(* CFC diagram, written out as Structured Text *)
(* KNX Sending interval *)
(* KNX Master *)
Interval(IN := Interval.Q);
_ADD9_OUT := BOOL_TO_INT(Interval.Q) + i;
i := _ADD9_OUT;
_GT15_OUT := i > 83;
_MOVE19_OUT := MOVE(EN := _GT15_OUT, IN := 0, ENO => _MOVE19_ENO);
IF _MOVE19_ENO THEN i := _MOVE19_OUT; END_IF;
KNX_master_1(I_Port := IoConfig_Globals.KNX_EIB_TP1_Interface, bPortKNX := 1);
STLV59_563.STLV59_A_563_KNX_Card_1_Status := KNX_master_1.sStatus = 'OK';
(* Rom 001 *)
(* RB601_V *)
(* RB601_HVAC *)
M1_001_001_RB601_V(bPortKNX := 1, dwIndex_DPT := 1, typDPT := typDPT);
_MOVE46_OUT := MOVE(EN := M1_001_001_RB601_V.xUpdate_PLC, IN := M1_001_001_RB601_V.xSwitch_OUT, ENO => _MOVE46_ENO);
IF _MOVE46_ENO THEN STLV59_563.STLV59_A_563_001.RB601_V := _MOVE46_OUT; END_IF;
M1_002_001_RB601_HVAC(bPortKNX := 1, dwIndex_DPT := 2, typDPT := typDPT);
_MOVE59_OUT := MOVE(EN := M1_002_001_RB601_HVAC.xUpdate_PLC, IN := M1_002_001_RB601_HVAC.xSwitch_OUT, ENO => _MOVE59_ENO);
IF _MOVE59_ENO THEN STLV59_563.STLV59_A_563_001.RB601_HVAC := _MOVE59_OUT; END_IF;
(* RT601_CT *)
(* RY601_CV *)
M1_003_001_RT601_CT(bPortKNX := 1, dwIndex_DPT := 3, typDPT := typDPT);
_MOVE72_OUT := MOVE(EN := M1_003_001_RT601_CT.xUpdate_PLC, IN := M1_003_001_RT601_CT.rValue_OUT, ENO => _MOVE72_ENO);
IF _MOVE72_ENO THEN STLV59_563.STLV59_A_563_001.RT601_CT := _MOVE72_OUT; END_IF;
M1_004_001_RY601_CV(bPortKNX := 1, dwIndex_DPT := 4, typDPT := typDPT);
_MOVE85_OUT := MOVE(EN := M1_004_001_RY601_CV.xUpdate_PLC, IN := M1_004_001_RY601_CV.rValue_OUT, ENO => _MOVE85_ENO);
IF _MOVE85_ENO THEN STLV59_563.STLV59_A_563_001.RY601_CV := _MOVE85_OUT; END_IF;
(* LH601_OP *)
(* LH601_CMD *)
M1_005_001_LH601_OP(bPortKNX := 1, dwIndex_DPT := 5, rValue_IN := STLV59_563.STLV59_A_563_001.LH601_OP, xUpdate_KNX := i = 0, typDPT := typDPT);
M1_006_001_LH601_CMD(bPortKNX := 1, dwIndex_DPT := 6, xSwitch_IN := STLV59_563.STLV59_A_563_001.LH601_CMD, xUpdate_KNX := i = 1, typDPT := typDPT);
(* LC601_OP *)
(* LC601_CMD *)
M1_007_001_LC601_OP(bPortKNX := 1, dwIndex_DPT := 7, rValue_IN := STLV59_563.STLV59_A_563_001.LC601_OP, xUpdate_KNX := i = 2, typDPT := typDPT);
M1_008_001_LC601_CMD(bPortKNX := 1, dwIndex_DPT := 8, xSwitch_IN := STLV59_563.STLV59_A_563_001.LC601_CMD, xUpdate_KNX := i = 3, typDPT := typDPT);
(* Rom 002 *)
(* RB601_V *)
(* RB602_V *)
M1_009_002_RB601_V(bPortKNX := 1, dwIndex_DPT := 9, typDPT := typDPT);
_MOVE163_OUT := MOVE(EN := M1_009_002_RB601_V.xUpdate_PLC, IN := M1_009_002_RB601_V.xSwitch_OUT, ENO => _MOVE163_ENO);
IF _MOVE163_ENO THEN STLV59_563.STLV59_A_563_002.RB601_V := _MOVE163_OUT; END_IF;
M1_0010_002_RB602_V(bPortKNX := 1, dwIndex_DPT := 10, typDPT := typDPT);
_MOVE176_OUT := MOVE(EN := M1_0010_002_RB602_V.xUpdate_PLC, IN := M1_0010_002_RB602_V.xSwitch_OUT, ENO => _MOVE176_ENO);
IF _MOVE176_ENO THEN STLV59_563.STLV59_A_563_002.RB602_V := _MOVE176_OUT; END_IF;
(* RB601_HVAC *)
(* RB602_HVAC *)
M1_011_002_RB601_HVAC(bPortKNX := 1, dwIndex_DPT := 11, typDPT := typDPT);
_MOVE189_OUT := MOVE(EN := M1_011_002_RB601_HVAC.xUpdate_PLC, IN := M1_011_002_RB601_HVAC.xSwitch_OUT, ENO => _MOVE189_ENO);
IF _MOVE189_ENO THEN STLV59_563.STLV59_A_563_002.RB601_HVAC := _MOVE189_OUT; END_IF;
M1_012_002_RB602_HVAC(bPortKNX := 1, dwIndex_DPT := 12, typDPT := typDPT);
_MOVE202_OUT := MOVE(EN := M1_012_002_RB602_HVAC.xUpdate_PLC, IN := M1_012_002_RB602_HVAC.xSwitch_OUT, ENO => _MOVE202_ENO);
IF _MOVE202_ENO THEN STLV59_563.STLV59_A_563_002.RB602_HVAC := _MOVE202_OUT; END_IF;
(* RT601_CT *)
(* RY601_CV *)
M1_013_002_RT601_CT(bPortKNX := 1, dwIndex_DPT := 13, typDPT := typDPT);
_MOVE215_OUT := MOVE(EN := M1_013_002_RT601_CT.xUpdate_PLC, IN := M1_013_002_RT601_CT.rValue_OUT, ENO => _MOVE215_ENO);
IF _MOVE215_ENO THEN STLV59_563.STLV59_A_563_002.RT601_CT := _MOVE215_OUT; END_IF;
M1_014_002_RY601_CV(bPortKNX := 1, dwIndex_DPT := 14, typDPT := typDPT);
_MOVE228_OUT := MOVE(EN := M1_014_002_RY601_CV.xUpdate_PLC, IN := M1_014_002_RY601_CV.rValue_OUT, ENO => _MOVE228_ENO);
IF _MOVE228_ENO THEN STLV59_563.STLV59_A_563_002.RY601_CV := _MOVE228_OUT; END_IF;
(* LH601_OP *)
(* LH601_CMD *)
M1_015_002_LH601_OP(bPortKNX := 1, dwIndex_DPT := 15, rValue_IN := STLV59_563.STLV59_A_563_002.LH601_OP, xUpdate_KNX := i = 4, typDPT := typDPT);
M1_016_002_LH601_CMD(bPortKNX := 1, dwIndex_DPT := 16, xSwitch_IN := STLV59_563.STLV59_A_563_002.LH601_CMD, xUpdate_KNX := i = 5, typDPT := typDPT);
(* LC601_OP *)
(* LC601_CMD *)
M1_017_002_LC601_OP(bPortKNX := 1, dwIndex_DPT := 17, rValue_IN := STLV59_563.STLV59_A_563_002.LC601_OP, xUpdate_KNX := i = 6, typDPT := typDPT);
M1_018_002_LC601_CMD(bPortKNX := 1, dwIndex_DPT := 18, xSwitch_IN := STLV59_563.STLV59_A_563_002.LC601_CMD, xUpdate_KNX := i = 7, typDPT := typDPT);
(* Rom 003 *)
(* RB601_V *)
(* RB601_HVAC *)
M1_019_003_RB601_V(bPortKNX := 1, dwIndex_DPT := 19, typDPT := typDPT);
_MOVE306_OUT := MOVE(EN := M1_019_003_RB601_V.xUpdate_PLC, IN := M1_019_003_RB601_V.xSwitch_OUT, ENO => _MOVE306_ENO);
IF _MOVE306_ENO THEN STLV59_563.STLV59_A_563_003.RB601_V := _MOVE306_OUT; END_IF;
M1_020_003_RB601_HVAC(bPortKNX := 1, dwIndex_DPT := 20, typDPT := typDPT);
_MOVE319_OUT := MOVE(EN := M1_020_003_RB601_HVAC.xUpdate_PLC, IN := M1_020_003_RB601_HVAC.xSwitch_OUT, ENO => _MOVE319_ENO);
IF _MOVE319_ENO THEN STLV59_563.STLV59_A_563_003.RB601_HVAC := _MOVE319_OUT; END_IF;
(* RT601_CT *)
(* RT602_CT *)
M1_021_003_RT601_CT(bPortKNX := 1, dwIndex_DPT := 21, typDPT := typDPT);
_MOVE332_OUT := MOVE(EN := M1_021_003_RT601_CT.xUpdate_PLC, IN := M1_021_003_RT601_CT.rValue_OUT, ENO => _MOVE332_ENO);
IF _MOVE332_ENO THEN STLV59_563.STLV59_A_563_003.RT601_CT := _MOVE332_OUT; END_IF;
M1_022_003_RT602_CT(bPortKNX := 1, dwIndex_DPT := 22, typDPT := typDPT);
_MOVE345_OUT := MOVE(EN := M1_022_003_RT602_CT.xUpdate_PLC, IN := M1_022_003_RT602_CT.rValue_OUT, ENO => _MOVE345_ENO);
IF _MOVE345_ENO THEN STLV59_563.STLV59_A_563_003.RT602_CT := _MOVE345_OUT; END_IF;
(* RY601_CV *)
(* LH601_OP *)
M1_023_003_RY601_CV(bPortKNX := 1, dwIndex_DPT := 23, typDPT := typDPT);
_MOVE358_OUT := MOVE(EN := M1_023_003_RY601_CV.xUpdate_PLC, IN := M1_023_003_RY601_CV.rValue_OUT, ENO => _MOVE358_ENO);
IF _MOVE358_ENO THEN STLV59_563.STLV59_A_563_003.RY601_CV := _MOVE358_OUT; END_IF;
M1_024_003_LH601_OP(bPortKNX := 1, dwIndex_DPT := 24, rValue_IN := STLV59_563.STLV59_A_563_003.LH601_OP, xUpdate_KNX := i = 8, typDPT := typDPT);
(* LH601_CMD *)
(* LC601_OP *)
M1_025_003_LH601_CMD(bPortKNX := 1, dwIndex_DPT := 25, xSwitch_IN := STLV59_563.STLV59_A_563_003.LH601_CMD, xUpdate_KNX := i = 9, typDPT := typDPT);
M1_026_003_LC601_OP(bPortKNX := 1, dwIndex_DPT := 26, rValue_IN := STLV59_563.STLV59_A_563_003.LC601_OP, xUpdate_KNX := i = 10, typDPT := typDPT);
(* LC601_CMD *)
M1_027_003_LC601_CMD(bPortKNX := 1, dwIndex_DPT := 27, xSwitch_IN := STLV59_563.STLV59_A_563_003.LC601_CMD, xUpdate_KNX := i = 11, typDPT := typDPT);
(* Rom 004 *)
(* RB601_V *)
(* RB601_HVAC *)
M1_028_004_RB601_V(bPortKNX := 1, dwIndex_DPT := 28, typDPT := typDPT);
_MOVE436_OUT := MOVE(EN := M1_028_004_RB601_V.xUpdate_PLC, IN := M1_028_004_RB601_V.xSwitch_OUT, ENO => _MOVE436_ENO);
IF _MOVE436_ENO THEN STLV59_563.STLV59_A_563_004.RB601_V := _MOVE436_OUT; END_IF;
M1_029_004_RB601_HVAC(bPortKNX := 1, dwIndex_DPT := 29, typDPT := typDPT);
_MOVE449_OUT := MOVE(EN := M1_029_004_RB601_HVAC.xUpdate_PLC, IN := M1_029_004_RB601_HVAC.xSwitch_OUT, ENO => _MOVE449_ENO);
IF _MOVE449_ENO THEN STLV59_563.STLV59_A_563_004.RB601_HVAC := _MOVE449_OUT; END_IF;
(* RT601_CT *)
(* RY601_CV *)
M1_030_004_RT601_CT(bPortKNX := 1, dwIndex_DPT := 30, typDPT := typDPT);
_MOVE462_OUT := MOVE(EN := M1_030_004_RT601_CT.xUpdate_PLC, IN := M1_030_004_RT601_CT.rValue_OUT, ENO => _MOVE462_ENO);
IF _MOVE462_ENO THEN STLV59_563.STLV59_A_563_004.RT601_CT := _MOVE462_OUT; END_IF;
M1_031_004_RY601_CV(bPortKNX := 1, dwIndex_DPT := 31, typDPT := typDPT);
_MOVE475_OUT := MOVE(EN := M1_031_004_RY601_CV.xUpdate_PLC, IN := M1_031_004_RY601_CV.rValue_OUT, ENO => _MOVE475_ENO);
IF _MOVE475_ENO THEN STLV59_563.STLV59_A_563_004.RY601_CV := _MOVE475_OUT; END_IF;
(* RY602_CV *)
(* LH601_OP *)
M1_032_004_RY602_CV(bPortKNX := 1, dwIndex_DPT := 32, typDPT := typDPT);
_MOVE488_OUT := MOVE(EN := M1_032_004_RY602_CV.xUpdate_PLC, IN := M1_032_004_RY602_CV.rValue_OUT, ENO => _MOVE488_ENO);
IF _MOVE488_ENO THEN STLV59_563.STLV59_A_563_004.RY602_CV := _MOVE488_OUT; END_IF;
M1_033_004_LH601_OP(bPortKNX := 1, dwIndex_DPT := 33, rValue_IN := STLV59_563.STLV59_A_563_004.LH601_OP, xUpdate_KNX := i = 12, typDPT := typDPT);
(* LH601_CMD *)
(* LC601_OP *)
M1_034_004_LH601_CMD(bPortKNX := 1, dwIndex_DPT := 34, xSwitch_IN := STLV59_563.STLV59_A_563_004.LH601_CMD, xUpdate_KNX := i = 13, typDPT := typDPT);
M1_035_004_LC601_OP(bPortKNX := 1, dwIndex_DPT := 35, rValue_IN := STLV59_563.STLV59_A_563_004.LC601_OP, xUpdate_KNX := i = 14, typDPT := typDPT);
(* LC601_CMD *)
M1_036_004_LC601_CMD(bPortKNX := 1, dwIndex_DPT := 36, xSwitch_IN := STLV59_563.STLV59_A_563_004.LC601_CMD, xUpdate_KNX := i = 15, typDPT := typDPT);
(* Rom 005 *)
(* RB601_V *)
(* RB601_HVAC *)
M1_037_005_RB601_V(bPortKNX := 1, dwIndex_DPT := 37, typDPT := typDPT);
_MOVE566_OUT := MOVE(EN := M1_037_005_RB601_V.xUpdate_PLC, IN := M1_037_005_RB601_V.xSwitch_OUT, ENO => _MOVE566_ENO);
IF _MOVE566_ENO THEN STLV59_563.STLV59_A_563_005.RB601_V := _MOVE566_OUT; END_IF;
M1_038_005_RB601_HVAC(bPortKNX := 1, dwIndex_DPT := 38, typDPT := typDPT);
_MOVE579_OUT := MOVE(EN := M1_038_005_RB601_HVAC.xUpdate_PLC, IN := M1_038_005_RB601_HVAC.xSwitch_OUT, ENO => _MOVE579_ENO);
IF _MOVE579_ENO THEN STLV59_563.STLV59_A_563_005.RB601_HVAC := _MOVE579_OUT; END_IF;
(* RT601_CT *)
(* RY601_CV *)
M1_039_005_RT601_CT(bPortKNX := 1, dwIndex_DPT := 39, typDPT := typDPT);
_MOVE592_OUT := MOVE(EN := M1_039_005_RT601_CT.xUpdate_PLC, IN := M1_039_005_RT601_CT.rValue_OUT, ENO => _MOVE592_ENO);
IF _MOVE592_ENO THEN STLV59_563.STLV59_A_563_005.RT601_CT := _MOVE592_OUT; END_IF;
M1_040_005_RY601_CV(bPortKNX := 1, dwIndex_DPT := 40, typDPT := typDPT);
_MOVE605_OUT := MOVE(EN := M1_040_005_RY601_CV.xUpdate_PLC, IN := M1_040_005_RY601_CV.rValue_OUT, ENO => _MOVE605_ENO);
IF _MOVE605_ENO THEN STLV59_563.STLV59_A_563_005.RY601_CV := _MOVE605_OUT; END_IF;
(* LH601_OP *)
(* LH602_OP *)
M1_041_005_LH601_OP(bPortKNX := 1, dwIndex_DPT := 41, rValue_IN := STLV59_563.STLV59_A_563_005.LH601_OP, xUpdate_KNX := i = 16, typDPT := typDPT);
M1_042_005_LH602_OP(bPortKNX := 1, dwIndex_DPT := 42, rValue_IN := STLV59_563.STLV59_A_563_005.LH602_OP, xUpdate_KNX := i = 17, typDPT := typDPT);
(* LH601_CMD *)
(* LC601_OP *)
M1_043_005_LH601_CMD(bPortKNX := 1, dwIndex_DPT := 43, xSwitch_IN := STLV59_563.STLV59_A_563_005.LH601_CMD, xUpdate_KNX := i = 18, typDPT := typDPT);
M1_044_005_LC601_OP(bPortKNX := 1, dwIndex_DPT := 44, rValue_IN := STLV59_563.STLV59_A_563_005.LC601_OP, xUpdate_KNX := i = 19, typDPT := typDPT);
(* LC601_CMD *)
M1_045_005_LC601_CMD(bPortKNX := 1, dwIndex_DPT := 45, xSwitch_IN := STLV59_563.STLV59_A_563_005.LC601_CMD, xUpdate_KNX := i = 20, typDPT := typDPT);
(* Rom 006 *)
(* RB601_V *)
(* RB601_HVAC *)
M1_046_006_RB601_V(bPortKNX := 1, dwIndex_DPT := 46, typDPT := typDPT);
_MOVE699_OUT := MOVE(EN := M1_046_006_RB601_V.xUpdate_PLC, IN := M1_046_006_RB601_V.xSwitch_OUT, ENO => _MOVE699_ENO);
IF _MOVE699_ENO THEN STLV59_563.STLV59_A_563_006.RB601_V := _MOVE699_OUT; END_IF;
M1_047_006_RB601_HVAC(bPortKNX := 1, dwIndex_DPT := 47, typDPT := typDPT);
_MOVE712_OUT := MOVE(EN := M1_047_006_RB601_HVAC.xUpdate_PLC, IN := M1_047_006_RB601_HVAC.xSwitch_OUT, ENO => _MOVE712_ENO);
IF _MOVE712_ENO THEN STLV59_563.STLV59_A_563_006.RB601_HVAC := _MOVE712_OUT; END_IF;
(* RT601_CT *)
(* RY601_CV *)
M1_048_006_RT601_CT(bPortKNX := 1, dwIndex_DPT := 48, typDPT := typDPT);
_MOVE725_OUT := MOVE(EN := M1_048_006_RT601_CT.xUpdate_PLC, IN := M1_048_006_RT601_CT.rValue_OUT, ENO => _MOVE725_ENO);
IF _MOVE725_ENO THEN STLV59_563.STLV59_A_563_006.RT601_CT := _MOVE725_OUT; END_IF;
M1_049_006_RY601_CV(bPortKNX := 1, dwIndex_DPT := 49, typDPT := typDPT);
_MOVE738_OUT := MOVE(EN := M1_049_006_RY601_CV.xUpdate_PLC, IN := M1_049_006_RY601_CV.rValue_OUT, ENO => _MOVE738_ENO);
IF _MOVE738_ENO THEN STLV59_563.STLV59_A_563_006.RY601_CV := _MOVE738_OUT; END_IF;
(* LH601_OP *)
(* LH601_CMD *)
M1_050_006_LH601_OP(bPortKNX := 1, dwIndex_DPT := 50, rValue_IN := STLV59_563.STLV59_A_563_006.LH601_OP, xUpdate_KNX := i = 21, typDPT := typDPT);
M1_051_006_LH601_CMD(bPortKNX := 1, dwIndex_DPT := 51, xSwitch_IN := STLV59_563.STLV59_A_563_006.LH601_CMD, xUpdate_KNX := i = 22, typDPT := typDPT);
(* LH602_CMD *)
(* LC601_OP *)
M1_052_006_LH602_CMD(bPortKNX := 1, dwIndex_DPT := 52, xSwitch_IN := STLV59_563.STLV59_A_563_006.LH602_CMD, xUpdate_KNX := i = 23, typDPT := typDPT);
M1_053_006_LC601_OP(bPortKNX := 1, dwIndex_DPT := 53, rValue_IN := STLV59_563.STLV59_A_563_006.LC601_OP, xUpdate_KNX := i = 24, typDPT := typDPT);
(* LC601_CMD *)
M1_054_006_LC601_CMD(bPortKNX := 1, dwIndex_DPT := 54, xSwitch_IN := STLV59_563.STLV59_A_563_006.LC601_CMD, xUpdate_KNX := i = 25, typDPT := typDPT);
(* Rom 007 *)
(* RB601_V *)
(* RB601_HVAC *)
M1_055_007_RB601_V(bPortKNX := 1, dwIndex_DPT := 55, typDPT := typDPT);
_MOVE832_OUT := MOVE(EN := M1_055_007_RB601_V.xUpdate_PLC, IN := M1_055_007_RB601_V.xSwitch_OUT, ENO => _MOVE832_ENO);
IF _MOVE832_ENO THEN STLV59_563.STLV59_A_563_007.RB601_V := _MOVE832_OUT; END_IF;
M1_056_007_RB601_HVAC(bPortKNX := 1, dwIndex_DPT := 56, typDPT := typDPT);
_MOVE845_OUT := MOVE(EN := M1_056_007_RB601_HVAC.xUpdate_PLC, IN := M1_056_007_RB601_HVAC.xSwitch_OUT, ENO => _MOVE845_ENO);
IF _MOVE845_ENO THEN STLV59_563.STLV59_A_563_007.RB601_HVAC := _MOVE845_OUT; END_IF;
(* RT601_CT *)
(* RY601_CV *)
M1_057_007_RT601_CT(bPortKNX := 1, dwIndex_DPT := 57, typDPT := typDPT);
_MOVE858_OUT := MOVE(EN := M1_057_007_RT601_CT.xUpdate_PLC, IN := M1_057_007_RT601_CT.rValue_OUT, ENO => _MOVE858_ENO);
IF _MOVE858_ENO THEN STLV59_563.STLV59_A_563_007.RT601_CT := _MOVE858_OUT; END_IF;
M1_058_007_RY601_CV(bPortKNX := 1, dwIndex_DPT := 58, typDPT := typDPT);
_MOVE871_OUT := MOVE(EN := M1_058_007_RY601_CV.xUpdate_PLC, IN := M1_058_007_RY601_CV.rValue_OUT, ENO => _MOVE871_ENO);
IF _MOVE871_ENO THEN STLV59_563.STLV59_A_563_007.RY601_CV := _MOVE871_OUT; END_IF;
(* LH601_OP *)
(* LH601_CMD *)
M1_059_007_LH601_OP(bPortKNX := 1, dwIndex_DPT := 59, rValue_IN := STLV59_563.STLV59_A_563_007.LH601_OP, xUpdate_KNX := i = 26, typDPT := typDPT);
M1_060_007_LH601_CMD(bPortKNX := 1, dwIndex_DPT := 60, xSwitch_IN := STLV59_563.STLV59_A_563_007.LH601_CMD, xUpdate_KNX := i = 27, typDPT := typDPT);
(* LC601_OP *)
(* LC602_OP *)
M1_061_007_LC601_OP(bPortKNX := 1, dwIndex_DPT := 61, rValue_IN := STLV59_563.STLV59_A_563_007.LC601_OP, xUpdate_KNX := i = 28, typDPT := typDPT);
M1_062_007_LC602_OP(bPortKNX := 1, dwIndex_DPT := 62, rValue_IN := STLV59_563.STLV59_A_563_007.LC602_OP, xUpdate_KNX := i = 29, typDPT := typDPT);
(* LC601_CMD *)
M1_063_007_LC601_CMD(bPortKNX := 1, dwIndex_DPT := 63, xSwitch_IN := STLV59_563.STLV59_A_563_007.LC601_CMD, xUpdate_KNX := i = 30, typDPT := typDPT);
(* Rom 008 *)
(* RB601_V *)
(* RB601_HVAC *)
M1_064_008_RB601_V(bPortKNX := 1, dwIndex_DPT := 64, typDPT := typDPT);
_MOVE965_OUT := MOVE(EN := M1_064_008_RB601_V.xUpdate_PLC, IN := M1_064_008_RB601_V.xSwitch_OUT, ENO => _MOVE965_ENO);
IF _MOVE965_ENO THEN STLV59_563.STLV59_A_563_008.RB601_V := _MOVE965_OUT; END_IF;
M1_065_008_RB601_HVAC(bPortKNX := 1, dwIndex_DPT := 65, typDPT := typDPT);
_MOVE978_OUT := MOVE(EN := M1_065_008_RB601_HVAC.xUpdate_PLC, IN := M1_065_008_RB601_HVAC.xSwitch_OUT, ENO => _MOVE978_ENO);
IF _MOVE978_ENO THEN STLV59_563.STLV59_A_563_008.RB601_HVAC := _MOVE978_OUT; END_IF;
(* RT601_CT *)
(* RY601_CV *)
M1_066_008_RT601_CT(bPortKNX := 1, dwIndex_DPT := 66, typDPT := typDPT);
_MOVE991_OUT := MOVE(EN := M1_066_008_RT601_CT.xUpdate_PLC, IN := M1_066_008_RT601_CT.rValue_OUT, ENO => _MOVE991_ENO);
IF _MOVE991_ENO THEN STLV59_563.STLV59_A_563_008.RT601_CT := _MOVE991_OUT; END_IF;
M1_067_008_RY601_CV(bPortKNX := 1, dwIndex_DPT := 67, typDPT := typDPT);
_MOVE1004_OUT := MOVE(EN := M1_067_008_RY601_CV.xUpdate_PLC, IN := M1_067_008_RY601_CV.rValue_OUT, ENO => _MOVE1004_ENO);
IF _MOVE1004_ENO THEN STLV59_563.STLV59_A_563_008.RY601_CV := _MOVE1004_OUT; END_IF;
(* LH601_OP *)
(* LH601_CMD *)
M1_068_008_LH601_OP(bPortKNX := 1, dwIndex_DPT := 68, rValue_IN := STLV59_563.STLV59_A_563_008.LH601_OP, xUpdate_KNX := i = 31, typDPT := typDPT);
M1_069_008_LH601_CMD(bPortKNX := 1, dwIndex_DPT := 69, xSwitch_IN := STLV59_563.STLV59_A_563_008.LH601_CMD, xUpdate_KNX := i = 32, typDPT := typDPT);
(* LC601_OP *)
(* LC601_CMD *)
M1_070_008_LC601_OP(bPortKNX := 1, dwIndex_DPT := 70, rValue_IN := STLV59_563.STLV59_A_563_008.LC601_OP, xUpdate_KNX := i = 33, typDPT := typDPT);
M1_071_008_LC601_CMD(bPortKNX := 1, dwIndex_DPT := 71, xSwitch_IN := STLV59_563.STLV59_A_563_008.LC601_CMD, xUpdate_KNX := i = 34, typDPT := typDPT);
(* LC602_CMD *)
M1_072_008_LC602_CMD(bPortKNX := 1, dwIndex_DPT := 72, xSwitch_IN := STLV59_563.STLV59_A_563_008.LC602_CMD, xUpdate_KNX := i = 35, typDPT := typDPT);
(* Rom 009 *)
(* RB601_V *)
(* RB601_HVAC *)
M1_073_009_RB601_V(bPortKNX := 1, dwIndex_DPT := 73, typDPT := typDPT);
_MOVE1098_OUT := MOVE(EN := M1_073_009_RB601_V.xUpdate_PLC, IN := M1_073_009_RB601_V.xSwitch_OUT, ENO => _MOVE1098_ENO);
IF _MOVE1098_ENO THEN STLV59_563.STLV59_A_563_009.RB601_V := _MOVE1098_OUT; END_IF;
M1_074_009_RB601_HVAC(bPortKNX := 1, dwIndex_DPT := 74, typDPT := typDPT);
_MOVE1111_OUT := MOVE(EN := M1_074_009_RB601_HVAC.xUpdate_PLC, IN := M1_074_009_RB601_HVAC.xSwitch_OUT, ENO => _MOVE1111_ENO);
IF _MOVE1111_ENO THEN STLV59_563.STLV59_A_563_009.RB601_HVAC := _MOVE1111_OUT; END_IF;
(* RT601_CT *)
(* RT602_CT *)
M1_075_009_RT601_CT(bPortKNX := 1, dwIndex_DPT := 75, typDPT := typDPT);
_MOVE1124_OUT := MOVE(EN := M1_075_009_RT601_CT.xUpdate_PLC, IN := M1_075_009_RT601_CT.rValue_OUT, ENO => _MOVE1124_ENO);
IF _MOVE1124_ENO THEN STLV59_563.STLV59_A_563_009.RT601_CT := _MOVE1124_OUT; END_IF;
M1_076_009_RT602_CT(bPortKNX := 1, dwIndex_DPT := 76, typDPT := typDPT);
_MOVE1137_OUT := MOVE(EN := M1_076_009_RT602_CT.xUpdate_PLC, IN := M1_076_009_RT602_CT.rValue_OUT, ENO => _MOVE1137_ENO);
IF _MOVE1137_ENO THEN STLV59_563.STLV59_A_563_009.RT602_CT := _MOVE1137_OUT; END_IF;
(* RY601_CV *)
(* LH601_OP *)
M1_077_009_RY601_CV(bPortKNX := 1, dwIndex_DPT := 77, typDPT := typDPT);
_MOVE1150_OUT := MOVE(EN := M1_077_009_RY601_CV.xUpdate_PLC, IN := M1_077_009_RY601_CV.rValue_OUT, ENO => _MOVE1150_ENO);
IF _MOVE1150_ENO THEN STLV59_563.STLV59_A_563_009.RY601_CV := _MOVE1150_OUT; END_IF;
M1_078_009_LH601_OP(bPortKNX := 1, dwIndex_DPT := 78, rValue_IN := STLV59_563.STLV59_A_563_009.LH601_OP, xUpdate_KNX := i = 36, typDPT := typDPT);
(* LH602_OP *)
(* LH601_CMD *)
M1_079_009_LH602_OP(bPortKNX := 1, dwIndex_DPT := 79, rValue_IN := STLV59_563.STLV59_A_563_009.LH602_OP, xUpdate_KNX := i = 37, typDPT := typDPT);
M1_080_009_LH601_CMD(bPortKNX := 1, dwIndex_DPT := 80, xSwitch_IN := STLV59_563.STLV59_A_563_009.LH601_CMD, xUpdate_KNX := i = 38, typDPT := typDPT);
(* LC601_OP *)
(* LC601_CMD *)
M1_081_009_LC601_OP(bPortKNX := 1, dwIndex_DPT := 81, rValue_IN := STLV59_563.STLV59_A_563_009.LC601_OP, xUpdate_KNX := i = 39, typDPT := typDPT);
M1_082_009_LC601_CMD(bPortKNX := 1, dwIndex_DPT := 82, xSwitch_IN := STLV59_563.STLV59_A_563_009.LC601_CMD, xUpdate_KNX := i = 40, typDPT := typDPT);
(* Rom 010 *)
(* RB601_V *)
(* RB601_HVAC *)
M1_083_010_RB601_V(bPortKNX := 1, dwIndex_DPT := 83, typDPT := typDPT);
_MOVE1244_OUT := MOVE(EN := M1_083_010_RB601_V.xUpdate_PLC, IN := M1_083_010_RB601_V.xSwitch_OUT, ENO => _MOVE1244_ENO);
IF _MOVE1244_ENO THEN STLV59_563.STLV59_A_563_010.RB601_V := _MOVE1244_OUT; END_IF;
M1_084_010_RB601_HVAC(bPortKNX := 1, dwIndex_DPT := 84, typDPT := typDPT);
_MOVE1257_OUT := MOVE(EN := M1_084_010_RB601_HVAC.xUpdate_PLC, IN := M1_084_010_RB601_HVAC.xSwitch_OUT, ENO => _MOVE1257_ENO);
IF _MOVE1257_ENO THEN STLV59_563.STLV59_A_563_010.RB601_HVAC := _MOVE1257_OUT; END_IF;
(* RT601_CT *)
(* RT602_CT *)
M1_085_010_RT601_CT(bPortKNX := 1, dwIndex_DPT := 85, typDPT := typDPT);
_MOVE1270_OUT := MOVE(EN := M1_085_010_RT601_CT.xUpdate_PLC, IN := M1_085_010_RT601_CT.rValue_OUT, ENO => _MOVE1270_ENO);
IF _MOVE1270_ENO THEN STLV59_563.STLV59_A_563_010.RT601_CT := _MOVE1270_OUT; END_IF;
M1_086_010_RT602_CT(bPortKNX := 1, dwIndex_DPT := 86, typDPT := typDPT);
_MOVE1283_OUT := MOVE(EN := M1_086_010_RT602_CT.xUpdate_PLC, IN := M1_086_010_RT602_CT.rValue_OUT, ENO => _MOVE1283_ENO);
IF _MOVE1283_ENO THEN STLV59_563.STLV59_A_563_010.RT602_CT := _MOVE1283_OUT; END_IF;
(* RY601_CV *)
(* LH601_OP *)
M1_087_010_RY601_CV(bPortKNX := 1, dwIndex_DPT := 87, typDPT := typDPT);
_MOVE1296_OUT := MOVE(EN := M1_087_010_RY601_CV.xUpdate_PLC, IN := M1_087_010_RY601_CV.rValue_OUT, ENO => _MOVE1296_ENO);
IF _MOVE1296_ENO THEN STLV59_563.STLV59_A_563_010.RY601_CV := _MOVE1296_OUT; END_IF;
M1_088_010_LH601_OP(bPortKNX := 1, dwIndex_DPT := 88, rValue_IN := STLV59_563.STLV59_A_563_010.LH601_OP, xUpdate_KNX := i = 41, typDPT := typDPT);
(* LH601_CMD *)
(* LH602_CMD *)
M1_089_010_LH601_CMD(bPortKNX := 1, dwIndex_DPT := 89, xSwitch_IN := STLV59_563.STLV59_A_563_010.LH601_CMD, xUpdate_KNX := i = 42, typDPT := typDPT);
M1_090_010_LH602_CMD(bPortKNX := 1, dwIndex_DPT := 90, xSwitch_IN := STLV59_563.STLV59_A_563_010.LH602_CMD, xUpdate_KNX := i = 43, typDPT := typDPT);
(* LC601_OP *)
(* LC601_CMD *)
M1_091_010_LC601_OP(bPortKNX := 1, dwIndex_DPT := 91, rValue_IN := STLV59_563.STLV59_A_563_010.LC601_OP, xUpdate_KNX := i = 44, typDPT := typDPT);
M1_092_010_LC601_CMD(bPortKNX := 1, dwIndex_DPT := 92, xSwitch_IN := STLV59_563.STLV59_A_563_010.LC601_CMD, xUpdate_KNX := i = 45, typDPT := typDPT);
(* Rom 011 *)
(* RB601_V *)
(* RB601_HVAC *)
M1_093_011_RB601_V(bPortKNX := 1, dwIndex_DPT := 93, typDPT := typDPT);
_MOVE1390_OUT := MOVE(EN := M1_093_011_RB601_V.xUpdate_PLC, IN := M1_093_011_RB601_V.xSwitch_OUT, ENO => _MOVE1390_ENO);
IF _MOVE1390_ENO THEN STLV59_563.STLV59_A_563_011.RB601_V := _MOVE1390_OUT; END_IF;
M1_094_011_RB601_HVAC(bPortKNX := 1, dwIndex_DPT := 94, typDPT := typDPT);
_MOVE1403_OUT := MOVE(EN := M1_094_011_RB601_HVAC.xUpdate_PLC, IN := M1_094_011_RB601_HVAC.xSwitch_OUT, ENO => _MOVE1403_ENO);
IF _MOVE1403_ENO THEN STLV59_563.STLV59_A_563_011.RB601_HVAC := _MOVE1403_OUT; END_IF;
(* RT601_CT *)
(* RT602_CT *)
M1_095_011_RT601_CT(bPortKNX := 1, dwIndex_DPT := 95, typDPT := typDPT);
_MOVE1416_OUT := MOVE(EN := M1_095_011_RT601_CT.xUpdate_PLC, IN := M1_095_011_RT601_CT.rValue_OUT, ENO => _MOVE1416_ENO);
IF _MOVE1416_ENO THEN STLV59_563.STLV59_A_563_011.RT601_CT := _MOVE1416_OUT; END_IF;
M1_096_011_RT602_CT(bPortKNX := 1, dwIndex_DPT := 96, typDPT := typDPT);
_MOVE1429_OUT := MOVE(EN := M1_096_011_RT602_CT.xUpdate_PLC, IN := M1_096_011_RT602_CT.rValue_OUT, ENO => _MOVE1429_ENO);
IF _MOVE1429_ENO THEN STLV59_563.STLV59_A_563_011.RT602_CT := _MOVE1429_OUT; END_IF;
(* RY601_CV *)
(* LH601_OP *)
M1_097_011_RY601_CV(bPortKNX := 1, dwIndex_DPT := 97, typDPT := typDPT);
_MOVE1442_OUT := MOVE(EN := M1_097_011_RY601_CV.xUpdate_PLC, IN := M1_097_011_RY601_CV.rValue_OUT, ENO => _MOVE1442_ENO);
IF _MOVE1442_ENO THEN STLV59_563.STLV59_A_563_011.RY601_CV := _MOVE1442_OUT; END_IF;
M1_098_011_LH601_OP(bPortKNX := 1, dwIndex_DPT := 98, rValue_IN := STLV59_563.STLV59_A_563_011.LH601_OP, xUpdate_KNX := i = 46, typDPT := typDPT);
(* LH601_CMD *)
(* LC601_OP *)
M1_099_011_LH601_CMD(bPortKNX := 1, dwIndex_DPT := 99, xSwitch_IN := STLV59_563.STLV59_A_563_011.LH601_CMD, xUpdate_KNX := i = 47, typDPT := typDPT);
M1_100_011_LC601_OP(bPortKNX := 1, dwIndex_DPT := 100, rValue_IN := STLV59_563.STLV59_A_563_011.LC601_OP, xUpdate_KNX := i = 48, typDPT := typDPT);
(* LC602_OP *)
(* LC601_CMD *)
M1_101_011_LC602_OP(bPortKNX := 1, dwIndex_DPT := 101, rValue_IN := STLV59_563.STLV59_A_563_011.LC602_OP, xUpdate_KNX := i = 49, typDPT := typDPT);
M1_102_011_LC601_CMD(bPortKNX := 1, dwIndex_DPT := 102, xSwitch_IN := STLV59_563.STLV59_A_563_011.LC601_CMD, xUpdate_KNX := i = 50, typDPT := typDPT);
(* Rom 012 *)
(* RB601_V *)
(* RB601_HVAC *)
M1_103_012_RB601_V(bPortKNX := 1, dwIndex_DPT := 103, typDPT := typDPT);
_MOVE1536_OUT := MOVE(EN := M1_103_012_RB601_V.xUpdate_PLC, IN := M1_103_012_RB601_V.xSwitch_OUT, ENO => _MOVE1536_ENO);
IF _MOVE1536_ENO THEN STLV59_563.STLV59_A_563_012.RB601_V := _MOVE1536_OUT; END_IF;
M1_104_012_RB601_HVAC(bPortKNX := 1, dwIndex_DPT := 104, typDPT := typDPT);
_MOVE1549_OUT := MOVE(EN := M1_104_012_RB601_HVAC.xUpdate_PLC, IN := M1_104_012_RB601_HVAC.xSwitch_OUT, ENO => _MOVE1549_ENO);
IF _MOVE1549_ENO THEN STLV59_563.STLV59_A_563_012.RB601_HVAC := _MOVE1549_OUT; END_IF;
(* RT601_CT *)
(* RT602_CT *)
M1_105_012_RT601_CT(bPortKNX := 1, dwIndex_DPT := 105, typDPT := typDPT);
_MOVE1562_OUT := MOVE(EN := M1_105_012_RT601_CT.xUpdate_PLC, IN := M1_105_012_RT601_CT.rValue_OUT, ENO => _MOVE1562_ENO);
IF _MOVE1562_ENO THEN STLV59_563.STLV59_A_563_012.RT601_CT := _MOVE1562_OUT; END_IF;
M1_106_012_RT602_CT(bPortKNX := 1, dwIndex_DPT := 106, typDPT := typDPT);
_MOVE1575_OUT := MOVE(EN := M1_106_012_RT602_CT.xUpdate_PLC, IN := M1_106_012_RT602_CT.rValue_OUT, ENO => _MOVE1575_ENO);
IF _MOVE1575_ENO THEN STLV59_563.STLV59_A_563_012.RT602_CT := _MOVE1575_OUT; END_IF;
(* RY601_CV *)
(* LH601_OP *)
M1_107_012_RY601_CV(bPortKNX := 1, dwIndex_DPT := 107, typDPT := typDPT);
_MOVE1588_OUT := MOVE(EN := M1_107_012_RY601_CV.xUpdate_PLC, IN := M1_107_012_RY601_CV.rValue_OUT, ENO => _MOVE1588_ENO);
IF _MOVE1588_ENO THEN STLV59_563.STLV59_A_563_012.RY601_CV := _MOVE1588_OUT; END_IF;
M1_108_012_LH601_OP(bPortKNX := 1, dwIndex_DPT := 108, rValue_IN := STLV59_563.STLV59_A_563_012.LH601_OP, xUpdate_KNX := i = 51, typDPT := typDPT);
(* LH601_CMD *)
(* LC601_OP *)
M1_109_012_LH601_CMD(bPortKNX := 1, dwIndex_DPT := 109, xSwitch_IN := STLV59_563.STLV59_A_563_012.LH601_CMD, xUpdate_KNX := i = 52, typDPT := typDPT);
M1_110_012_LC601_OP(bPortKNX := 1, dwIndex_DPT := 110, rValue_IN := STLV59_563.STLV59_A_563_012.LC601_OP, xUpdate_KNX := i = 53, typDPT := typDPT);
(* LC601_CMD *)
(* LC602_CMD *)
M1_111_012_LC601_CMD(bPortKNX := 1, dwIndex_DPT := 111, xSwitch_IN := STLV59_563.STLV59_A_563_012.LC601_CMD, xUpdate_KNX := i = 54, typDPT := typDPT);
M1_112_012_LC602_CMD(bPortKNX := 1, dwIndex_DPT := 112, xSwitch_IN := STLV59_563.STLV59_A_563_012.LC602_CMD, xUpdate_KNX := i = 55, typDPT := typDPT);
(* Rom 013 *)
(* RB601_V *)
(* RB601_HVAC *)
M1_113_013_RB601_V(bPortKNX := 1, dwIndex_DPT := 113, typDPT := typDPT);
_MOVE1682_OUT := MOVE(EN := M1_113_013_RB601_V.xUpdate_PLC, IN := M1_113_013_RB601_V.xSwitch_OUT, ENO => _MOVE1682_ENO);
IF _MOVE1682_ENO THEN STLV59_563.STLV59_A_563_013.RB601_V := _MOVE1682_OUT; END_IF;
M1_114_013_RB601_HVAC(bPortKNX := 1, dwIndex_DPT := 114, typDPT := typDPT);
_MOVE1695_OUT := MOVE(EN := M1_114_013_RB601_HVAC.xUpdate_PLC, IN := M1_114_013_RB601_HVAC.xSwitch_OUT, ENO => _MOVE1695_ENO);
IF _MOVE1695_ENO THEN STLV59_563.STLV59_A_563_013.RB601_HVAC := _MOVE1695_OUT; END_IF;
(* RT601_CT *)
(* RT602_CT *)
M1_115_013_RT601_CT(bPortKNX := 1, dwIndex_DPT := 115, typDPT := typDPT);
_MOVE1708_OUT := MOVE(EN := M1_115_013_RT601_CT.xUpdate_PLC, IN := M1_115_013_RT601_CT.rValue_OUT, ENO => _MOVE1708_ENO);
IF _MOVE1708_ENO THEN STLV59_563.STLV59_A_563_013.RT601_CT := _MOVE1708_OUT; END_IF;
M1_116_013_RT602_CT(bPortKNX := 1, dwIndex_DPT := 116, typDPT := typDPT);
_MOVE1721_OUT := MOVE(EN := M1_116_013_RT602_CT.xUpdate_PLC, IN := M1_116_013_RT602_CT.rValue_OUT, ENO => _MOVE1721_ENO);
IF _MOVE1721_ENO THEN STLV59_563.STLV59_A_563_013.RT602_CT := _MOVE1721_OUT; END_IF;
(* RY601_CV *)
(* RY602_CV *)
M1_117_013_RY601_CV(bPortKNX := 1, dwIndex_DPT := 117, typDPT := typDPT);
_MOVE1734_OUT := MOVE(EN := M1_117_013_RY601_CV.xUpdate_PLC, IN := M1_117_013_RY601_CV.rValue_OUT, ENO => _MOVE1734_ENO);
IF _MOVE1734_ENO THEN STLV59_563.STLV59_A_563_013.RY601_CV := _MOVE1734_OUT; END_IF;
M1_118_013_RY602_CV(bPortKNX := 1, dwIndex_DPT := 118, typDPT := typDPT);
_MOVE1747_OUT := MOVE(EN := M1_118_013_RY602_CV.xUpdate_PLC, IN := M1_118_013_RY602_CV.rValue_OUT, ENO => _MOVE1747_ENO);
IF _MOVE1747_ENO THEN STLV59_563.STLV59_A_563_013.RY602_CV := _MOVE1747_OUT; END_IF;
(* LH601_OP *)
(* LH601_CMD *)
M1_119_013_LH601_OP(bPortKNX := 1, dwIndex_DPT := 119, rValue_IN := STLV59_563.STLV59_A_563_013.LH601_OP, xUpdate_KNX := i = 56, typDPT := typDPT);
M1_120_013_LH601_CMD(bPortKNX := 1, dwIndex_DPT := 120, xSwitch_IN := STLV59_563.STLV59_A_563_013.LH601_CMD, xUpdate_KNX := i = 57, typDPT := typDPT);
(* LC601_OP *)
(* LC601_CMD *)
M1_121_013_LC601_OP(bPortKNX := 1, dwIndex_DPT := 121, rValue_IN := STLV59_563.STLV59_A_563_013.LC601_OP, xUpdate_KNX := i = 58, typDPT := typDPT);
M1_122_013_LC601_CMD(bPortKNX := 1, dwIndex_DPT := 122, xSwitch_IN := STLV59_563.STLV59_A_563_013.LC601_CMD, xUpdate_KNX := i = 59, typDPT := typDPT);
(* Rom 014 *)
(* RB601_V *)
(* RB601_HVAC *)
M1_123_014_RB601_V(bPortKNX := 1, dwIndex_DPT := 123, typDPT := typDPT);
_MOVE1825_OUT := MOVE(EN := M1_123_014_RB601_V.xUpdate_PLC, IN := M1_123_014_RB601_V.xSwitch_OUT, ENO => _MOVE1825_ENO);
IF _MOVE1825_ENO THEN STLV59_563.STLV59_A_563_014.RB601_V := _MOVE1825_OUT; END_IF;
M1_124_014_RB601_HVAC(bPortKNX := 1, dwIndex_DPT := 124, typDPT := typDPT);
_MOVE1838_OUT := MOVE(EN := M1_124_014_RB601_HVAC.xUpdate_PLC, IN := M1_124_014_RB601_HVAC.xSwitch_OUT, ENO => _MOVE1838_ENO);
IF _MOVE1838_ENO THEN STLV59_563.STLV59_A_563_014.RB601_HVAC := _MOVE1838_OUT; END_IF;
(* RT601_CT *)
(* RT602_CT *)
M1_125_014_RT601_CT(bPortKNX := 1, dwIndex_DPT := 125, typDPT := typDPT);
_MOVE1851_OUT := MOVE(EN := M1_125_014_RT601_CT.xUpdate_PLC, IN := M1_125_014_RT601_CT.rValue_OUT, ENO => _MOVE1851_ENO);
IF _MOVE1851_ENO THEN STLV59_563.STLV59_A_563_014.RT601_CT := _MOVE1851_OUT; END_IF;
M1_126_014_RT602_CT(bPortKNX := 1, dwIndex_DPT := 126, typDPT := typDPT);
_MOVE1864_OUT := MOVE(EN := M1_126_014_RT602_CT.xUpdate_PLC, IN := M1_126_014_RT602_CT.rValue_OUT, ENO => _MOVE1864_ENO);
IF _MOVE1864_ENO THEN STLV59_563.STLV59_A_563_014.RT602_CT := _MOVE1864_OUT; END_IF;
(* RY601_CV *)
(* RY602_CV *)
M1_127_014_RY601_CV(bPortKNX := 1, dwIndex_DPT := 127, typDPT := typDPT);
_MOVE1877_OUT := MOVE(EN := M1_127_014_RY601_CV.xUpdate_PLC, IN := M1_127_014_RY601_CV.rValue_OUT, ENO => _MOVE1877_ENO);
IF _MOVE1877_ENO THEN STLV59_563.STLV59_A_563_014.RY601_CV := _MOVE1877_OUT; END_IF;
M1_128_014_RY602_CV(bPortKNX := 1, dwIndex_DPT := 128, typDPT := typDPT);
_MOVE1890_OUT := MOVE(EN := M1_128_014_RY602_CV.xUpdate_PLC, IN := M1_128_014_RY602_CV.rValue_OUT, ENO => _MOVE1890_ENO);
IF _MOVE1890_ENO THEN STLV59_563.STLV59_A_563_014.RY602_CV := _MOVE1890_OUT; END_IF;
(* LH601_OP *)
(* LH602_OP *)
M1_129_014_LH601_OP(bPortKNX := 1, dwIndex_DPT := 129, rValue_IN := STLV59_563.STLV59_A_563_014.LH601_OP, xUpdate_KNX := i = 60, typDPT := typDPT);
M1_130_014_LH602_OP(bPortKNX := 1, dwIndex_DPT := 130, rValue_IN := STLV59_563.STLV59_A_563_014.LH602_OP, xUpdate_KNX := i = 61, typDPT := typDPT);
(* LH601_CMD *)
(* LH602_CMD *)
M1_131_014_LH601_CMD(bPortKNX := 1, dwIndex_DPT := 131, xSwitch_IN := STLV59_563.STLV59_A_563_014.LH601_CMD, xUpdate_KNX := i = 62, typDPT := typDPT);
M1_132_014_LH602_CMD(bPortKNX := 1, dwIndex_DPT := 132, xSwitch_IN := STLV59_563.STLV59_A_563_014.LH602_CMD, xUpdate_KNX := i = 63, typDPT := typDPT);
(* LC601_OP *)
(* LC602_OP *)
M1_133_014_LC601_OP(bPortKNX := 1, dwIndex_DPT := 133, rValue_IN := STLV59_563.STLV59_A_563_014.LC601_OP, xUpdate_KNX := i = 64, typDPT := typDPT);
M1_134_014_LC602_OP(bPortKNX := 1, dwIndex_DPT := 134, rValue_IN := STLV59_563.STLV59_A_563_014.LC602_OP, xUpdate_KNX := i = 65, typDPT := typDPT);
(* LC601_CMD *)
(* LC602_CMD *)
M1_135_014_LC601_CMD(bPortKNX := 1, dwIndex_DPT := 135, xSwitch_IN := STLV59_563.STLV59_A_563_014.LC601_CMD, xUpdate_KNX := i = 66, typDPT := typDPT);
M1_136_014_LC602_CMD(bPortKNX := 1, dwIndex_DPT := 136, xSwitch_IN := STLV59_563.STLV59_A_563_014.LC602_CMD, xUpdate_KNX := i = 67, typDPT := typDPT);
(* Rom 015 *)
(* RB601_V *)
(* RB602_V *)
M1_137_015_RB601_V(bPortKNX := 1, dwIndex_DPT := 137, typDPT := typDPT);
_MOVE2032_OUT := MOVE(EN := M1_137_015_RB601_V.xUpdate_PLC, IN := M1_137_015_RB601_V.xSwitch_OUT, ENO => _MOVE2032_ENO);
IF _MOVE2032_ENO THEN STLV59_563.STLV59_A_563_015.RB601_V := _MOVE2032_OUT; END_IF;
M1_138_015_RB602_V(bPortKNX := 1, dwIndex_DPT := 138, typDPT := typDPT);
_MOVE2045_OUT := MOVE(EN := M1_138_015_RB602_V.xUpdate_PLC, IN := M1_138_015_RB602_V.xSwitch_OUT, ENO => _MOVE2045_ENO);
IF _MOVE2045_ENO THEN STLV59_563.STLV59_A_563_015.RB602_V := _MOVE2045_OUT; END_IF;
(* RB601_HVAC *)
(* RB602_HVAC *)
M1_139_015_RB601_HVAC(bPortKNX := 1, dwIndex_DPT := 139, typDPT := typDPT);
_MOVE2058_OUT := MOVE(EN := M1_139_015_RB601_HVAC.xUpdate_PLC, IN := M1_139_015_RB601_HVAC.xSwitch_OUT, ENO => _MOVE2058_ENO);
IF _MOVE2058_ENO THEN STLV59_563.STLV59_A_563_015.RB601_HVAC := _MOVE2058_OUT; END_IF;
M1_140_015_RB602_HVAC(bPortKNX := 1, dwIndex_DPT := 140, typDPT := typDPT);
_MOVE2071_OUT := MOVE(EN := M1_140_015_RB602_HVAC.xUpdate_PLC, IN := M1_140_015_RB602_HVAC.xSwitch_OUT, ENO => _MOVE2071_ENO);
IF _MOVE2071_ENO THEN STLV59_563.STLV59_A_563_015.RB602_HVAC := _MOVE2071_OUT; END_IF;
(* RT601_CT *)
(* RT602_CT *)
M1_141_015_RT601_CT(bPortKNX := 1, dwIndex_DPT := 141, typDPT := typDPT);
_MOVE2084_OUT := MOVE(EN := M1_141_015_RT601_CT.xUpdate_PLC, IN := M1_141_015_RT601_CT.rValue_OUT, ENO => _MOVE2084_ENO);
IF _MOVE2084_ENO THEN STLV59_563.STLV59_A_563_015.RT601_CT := _MOVE2084_OUT; END_IF;
M1_142_015_RT602_CT(bPortKNX := 1, dwIndex_DPT := 142, typDPT := typDPT);
_MOVE2097_OUT := MOVE(EN := M1_142_015_RT602_CT.xUpdate_PLC, IN := M1_142_015_RT602_CT.rValue_OUT, ENO => _MOVE2097_ENO);
IF _MOVE2097_ENO THEN STLV59_563.STLV59_A_563_015.RT602_CT := _MOVE2097_OUT; END_IF;
(* RY601_CV *)
(* RY602_CV *)
M1_143_015_RY601_CV(bPortKNX := 1, dwIndex_DPT := 143, typDPT := typDPT);
_MOVE2110_OUT := MOVE(EN := M1_143_015_RY601_CV.xUpdate_PLC, IN := M1_143_015_RY601_CV.rValue_OUT, ENO => _MOVE2110_ENO);
IF _MOVE2110_ENO THEN STLV59_563.STLV59_A_563_015.RY601_CV := _MOVE2110_OUT; END_IF;
M1_144_015_RY602_CV(bPortKNX := 1, dwIndex_DPT := 144, typDPT := typDPT);
_MOVE2123_OUT := MOVE(EN := M1_144_015_RY602_CV.xUpdate_PLC, IN := M1_144_015_RY602_CV.rValue_OUT, ENO => _MOVE2123_ENO);
IF _MOVE2123_ENO THEN STLV59_563.STLV59_A_563_015.RY602_CV := _MOVE2123_OUT; END_IF;
(* LH601_OP *)
(* LH602_OP *)
M1_145_015_LH601_OP(bPortKNX := 1, dwIndex_DPT := 145, rValue_IN := STLV59_563.STLV59_A_563_015.LH601_OP, xUpdate_KNX := i = 68, typDPT := typDPT);
M1_146_015_LH602_OP(bPortKNX := 1, dwIndex_DPT := 146, rValue_IN := STLV59_563.STLV59_A_563_015.LH602_OP, xUpdate_KNX := i = 69, typDPT := typDPT);
(* LH601_CMD *)
(* LH602_CMD *)
M1_147_015_LH601_CMD(bPortKNX := 1, dwIndex_DPT := 147, xSwitch_IN := STLV59_563.STLV59_A_563_015.LH601_CMD, xUpdate_KNX := i = 70, typDPT := typDPT);
M1_148_015_LH602_CMD(bPortKNX := 1, dwIndex_DPT := 148, xSwitch_IN := STLV59_563.STLV59_A_563_015.LH602_CMD, xUpdate_KNX := i = 71, typDPT := typDPT);
(* LC601_OP *)
(* LC602_OP *)
M1_149_015_LC601_OP(bPortKNX := 1, dwIndex_DPT := 149, rValue_IN := STLV59_563.STLV59_A_563_015.LC601_OP, xUpdate_KNX := i = 72, typDPT := typDPT);
M1_150_015_LC602_OP(bPortKNX := 1, dwIndex_DPT := 150, rValue_IN := STLV59_563.STLV59_A_563_015.LC602_OP, xUpdate_KNX := i = 73, typDPT := typDPT);
(* LC601_CMD *)
(* LC602_CMD *)
M1_151_015_LC601_CMD(bPortKNX := 1, dwIndex_DPT := 151, xSwitch_IN := STLV59_563.STLV59_A_563_015.LC601_CMD, xUpdate_KNX := i = 74, typDPT := typDPT);
M1_152_015_LC602_CMD(bPortKNX := 1, dwIndex_DPT := 152, xSwitch_IN := STLV59_563.STLV59_A_563_015.LC602_CMD, xUpdate_KNX := i = 75, typDPT := typDPT);
(* Rom 016 *)
(* RB601_V *)
(* RB602_V *)
M1_153_016_RB601_V(bPortKNX := 1, dwIndex_DPT := 153, typDPT := typDPT);
_MOVE2265_OUT := MOVE(EN := M1_153_016_RB601_V.xUpdate_PLC, IN := M1_153_016_RB601_V.xSwitch_OUT, ENO => _MOVE2265_ENO);
IF _MOVE2265_ENO THEN STLV59_563.STLV59_A_563_016.RB601_V := _MOVE2265_OUT; END_IF;
M1_154_016_RB602_V(bPortKNX := 1, dwIndex_DPT := 154, typDPT := typDPT);
_MOVE2278_OUT := MOVE(EN := M1_154_016_RB602_V.xUpdate_PLC, IN := M1_154_016_RB602_V.xSwitch_OUT, ENO => _MOVE2278_ENO);
IF _MOVE2278_ENO THEN STLV59_563.STLV59_A_563_016.RB602_V := _MOVE2278_OUT; END_IF;
(* RB601_HVAC *)
(* RB602_HVAC *)
M1_155_016_RB601_HVAC(bPortKNX := 1, dwIndex_DPT := 155, typDPT := typDPT);
_MOVE2291_OUT := MOVE(EN := M1_155_016_RB601_HVAC.xUpdate_PLC, IN := M1_155_016_RB601_HVAC.xSwitch_OUT, ENO => _MOVE2291_ENO);
IF _MOVE2291_ENO THEN STLV59_563.STLV59_A_563_016.RB601_HVAC := _MOVE2291_OUT; END_IF;
M1_156_016_RB602_HVAC(bPortKNX := 1, dwIndex_DPT := 156, typDPT := typDPT);
_MOVE2304_OUT := MOVE(EN := M1_156_016_RB602_HVAC.xUpdate_PLC, IN := M1_156_016_RB602_HVAC.xSwitch_OUT, ENO => _MOVE2304_ENO);
IF _MOVE2304_ENO THEN STLV59_563.STLV59_A_563_016.RB602_HVAC := _MOVE2304_OUT; END_IF;
(* RY601_CV *)
(* RY602_CV *)
M1_157_016_RY601_CV(bPortKNX := 1, dwIndex_DPT := 157, typDPT := typDPT);
_MOVE2317_OUT := MOVE(EN := M1_157_016_RY601_CV.xUpdate_PLC, IN := M1_157_016_RY601_CV.rValue_OUT, ENO => _MOVE2317_ENO);
IF _MOVE2317_ENO THEN STLV59_563.STLV59_A_563_016.RY601_CV := _MOVE2317_OUT; END_IF;
M1_158_016_RY602_CV(bPortKNX := 1, dwIndex_DPT := 158, typDPT := typDPT);
_MOVE2330_OUT := MOVE(EN := M1_158_016_RY602_CV.xUpdate_PLC, IN := M1_158_016_RY602_CV.rValue_OUT, ENO => _MOVE2330_ENO);
IF _MOVE2330_ENO THEN STLV59_563.STLV59_A_563_016.RY602_CV := _MOVE2330_OUT; END_IF;
(* LH601_OP *)
(* LH602_OP *)
M1_159_016_LH601_OP(bPortKNX := 1, dwIndex_DPT := 159, rValue_IN := STLV59_563.STLV59_A_563_016.LH601_OP, xUpdate_KNX := i = 76, typDPT := typDPT);
M1_160_016_LH602_OP(bPortKNX := 1, dwIndex_DPT := 160, rValue_IN := STLV59_563.STLV59_A_563_016.LH602_OP, xUpdate_KNX := i = 77, typDPT := typDPT);
(* LH601_CMD *)
(* LH602_CMD *)
M1_161_016_LH601_CMD(bPortKNX := 1, dwIndex_DPT := 161, xSwitch_IN := STLV59_563.STLV59_A_563_016.LH601_CMD, xUpdate_KNX := i = 78, typDPT := typDPT);
M1_162_016_LH602_CMD(bPortKNX := 1, dwIndex_DPT := 162, xSwitch_IN := STLV59_563.STLV59_A_563_016.LH602_CMD, xUpdate_KNX := i = 79, typDPT := typDPT);
(* LC601_OP *)
(* LC602_OP *)
M1_163_016_LC601_OP(bPortKNX := 1, dwIndex_DPT := 163, rValue_IN := STLV59_563.STLV59_A_563_016.LC601_OP, xUpdate_KNX := i = 80, typDPT := typDPT);
M1_164_016_LC602_OP(bPortKNX := 1, dwIndex_DPT := 164, rValue_IN := STLV59_563.STLV59_A_563_016.LC602_OP, xUpdate_KNX := i = 81, typDPT := typDPT);
(* LC601_CMD *)
(* LC602_CMD *)
M1_165_016_LC601_CMD(bPortKNX := 1, dwIndex_DPT := 165, xSwitch_IN := STLV59_563.STLV59_A_563_016.LC601_CMD, xUpdate_KNX := i = 82, typDPT := typDPT);
M1_166_016_LC602_CMD(bPortKNX := 1, dwIndex_DPT := 166, xSwitch_IN := STLV59_563.STLV59_A_563_016.LC602_CMD, xUpdate_KNX := i = 83, typDPT := typDPT);
END_PROGRAM

PROGRAM PRG_563_Romstyring
  VAR
    Rom_001 : fbRomtype_11111111;  (* 001 *)
    Rom_002 : fbRomtype_22111111;  (* 002 *)
    Rom_003 : fbRomtype_11211111;  (* 003 *)
    Rom_004 : fbRomtype_11121111;  (* 004 *)
    Rom_005 : fbRomtype_11112111;  (* 005 *)
    Rom_006 : fbRomtype_11111211;  (* 006 *)
    Rom_007 : fbRomtype_11111121;  (* 007 *)
    Rom_008 : fbRomtype_11111112;  (* 008 *)
    Rom_009 : fbRomtype_11212111;  (* 009 *)
    Rom_010 : fbRomtype_11211211;  (* 010 *)
    Rom_011 : fbRomtype_11211121;  (* 011 *)
    Rom_012 : fbRomtype_11211112;  (* 012 *)
    Rom_013 : fbRomtype_11221111;  (* 013 *)
    Rom_014 : fbRomtype_11222222;  (* 014 *)
    Rom_015 : fbRomtype_22222222;  (* 015 *)
    Rom_016 : fbRomtype_22022222;  (* 016 *)
  END_VAR

(* CFC diagram, written out as Structured Text *)
(* Rom 001 *)
Rom_001(RB601_HVAC := STLV59_563.STLV59_A_563_001.RB601_HVAC, RT601_CT := STLV59_563.STLV59_A_563_001.RT601_CT, RT601_SP_D := STLV59_563.STLV59_A_563_001.RT601_SP_D, RT601_SP_S := STLV59_563.STLV59_A_563_001.RT601_SP_S, RT601_SP_N := STLV59_563.STLV59_A_563_001.RT601_SP_N, RT601_SP_F := STLV59_563.STLV59_A_563_001.RT601_SP_F, OPM := STLV59_563.STLV59_A_563_001.OPM, RY601_CV := STLV59_563.STLV59_A_563_001.RY601_CV, RY601_SP := STLV59_563.STLV59_A_563_001.RY601_SP, RY601_MAN := STLV59_563.STLV59_A_563_001.RY601_MAN, LH601_MAN := STLV59_563.STLV59_A_563_001.LH601_MAN, LC601_SP := STLV59_563.STLV59_A_563_001.LC601_SP, LC601_MAN := STLV59_563.STLV59_A_563_001.LC601_MAN);
STLV59_563.STLV59_A_563_001.OPM_CV := Rom_001.OPM_CV;
STLV59_563.STLV59_A_563_001.RT601_CS := Rom_001.RT601_CS;
STLV59_563.STLV59_A_563_001.RY601_OP := Rom_001.RY601_OP;
STLV59_563.STLV59_A_563_001.LH601_OP := Rom_001.LH601_OP;
STLV59_563.STLV59_A_563_001.LH601_CMD := Rom_001.LH601_CMD;
STLV59_563.STLV59_A_563_001.LC601_OP := Rom_001.LC601_OP;
STLV59_563.STLV59_A_563_001.LC601_CMD := Rom_001.LC601_CMD;
(* Rom 002 *)
Rom_002(RB601_HVAC := STLV59_563.STLV59_A_563_002.RB601_HVAC, RB602_HVAC := STLV59_563.STLV59_A_563_002.RB602_HVAC, RT601_CT := STLV59_563.STLV59_A_563_002.RT601_CT, RT601_SP_D := STLV59_563.STLV59_A_563_002.RT601_SP_D, RT601_SP_S := STLV59_563.STLV59_A_563_002.RT601_SP_S, RT601_SP_N := STLV59_563.STLV59_A_563_002.RT601_SP_N, RT601_SP_F := STLV59_563.STLV59_A_563_002.RT601_SP_F, OPM := STLV59_563.STLV59_A_563_002.OPM, RY601_CV := STLV59_563.STLV59_A_563_002.RY601_CV, RY601_SP := STLV59_563.STLV59_A_563_002.RY601_SP, RY601_MAN := STLV59_563.STLV59_A_563_002.RY601_MAN, LH601_MAN := STLV59_563.STLV59_A_563_002.LH601_MAN, LC601_SP := STLV59_563.STLV59_A_563_002.LC601_SP, LC601_MAN := STLV59_563.STLV59_A_563_002.LC601_MAN);
STLV59_563.STLV59_A_563_002.RB600_HVAC := Rom_002.RB600_HVAC;
STLV59_563.STLV59_A_563_002.OPM_CV := Rom_002.OPM_CV;
STLV59_563.STLV59_A_563_002.RT601_CS := Rom_002.RT601_CS;
STLV59_563.STLV59_A_563_002.RY601_OP := Rom_002.RY601_OP;
STLV59_563.STLV59_A_563_002.LH601_OP := Rom_002.LH601_OP;
STLV59_563.STLV59_A_563_002.LH601_CMD := Rom_002.LH601_CMD;
STLV59_563.STLV59_A_563_002.LC601_OP := Rom_002.LC601_OP;
STLV59_563.STLV59_A_563_002.LC601_CMD := Rom_002.LC601_CMD;
(* Rom 003 *)
Rom_003(RB601_HVAC := STLV59_563.STLV59_A_563_003.RB601_HVAC, RT601_CT := STLV59_563.STLV59_A_563_003.RT601_CT, RT602_CT := STLV59_563.STLV59_A_563_003.RT602_CT, RT600_SP_D := STLV59_563.STLV59_A_563_003.RT600_SP_D, RT600_SP_S := STLV59_563.STLV59_A_563_003.RT600_SP_S, RT600_SP_N := STLV59_563.STLV59_A_563_003.RT600_SP_N, RT600_SP_F := STLV59_563.STLV59_A_563_003.RT600_SP_F, OPM := STLV59_563.STLV59_A_563_003.OPM, RY601_CV := STLV59_563.STLV59_A_563_003.RY601_CV, RY601_SP := STLV59_563.STLV59_A_563_003.RY601_SP, RY601_MAN := STLV59_563.STLV59_A_563_003.RY601_MAN, LH600_MAN := STLV59_563.STLV59_A_563_003.LH601_MAN, LC600_SP := STLV59_563.STLV59_A_563_003.LC601_SP, LC600_MAN := STLV59_563.STLV59_A_563_003.LC601_MAN);
STLV59_563.STLV59_A_563_003.OPM_CV := Rom_003.OPM_CV;
STLV59_563.STLV59_A_563_003.RT600_CT := Rom_003.RT600_CT;
STLV59_563.STLV59_A_563_003.RT600_CS := Rom_003.RT600_CS;
STLV59_563.STLV59_A_563_003.RY601_OP := Rom_003.RY601_OP;
STLV59_563.STLV59_A_563_003.LH601_OP := Rom_003.LH601_OP;
STLV59_563.STLV59_A_563_003.LH601_CMD := Rom_003.LH601_CMD;
STLV59_563.STLV59_A_563_003.LC601_OP := Rom_003.LC601_OP;
STLV59_563.STLV59_A_563_003.LC601_CMD := Rom_003.LC601_CMD;
(* Rom 004 *)
Rom_004(RB601_HVAC := STLV59_563.STLV59_A_563_004.RB601_HVAC, RT601_CT := STLV59_563.STLV59_A_563_004.RT601_CT, RT601_SP_D := STLV59_563.STLV59_A_563_004.RT601_SP_D, RT601_SP_S := STLV59_563.STLV59_A_563_004.RT601_SP_S, RT601_SP_N := STLV59_563.STLV59_A_563_004.RT601_SP_N, RT601_SP_F := STLV59_563.STLV59_A_563_004.RT601_SP_F, OPM := STLV59_563.STLV59_A_563_004.OPM, RY601_CV := STLV59_563.STLV59_A_563_004.RY601_CV, RY602_CV := STLV59_563.STLV59_A_563_004.RY602_CV, RY600_SP := STLV59_563.STLV59_A_563_004.RY600_SP, RY600_MAN := STLV59_563.STLV59_A_563_004.RY600_MAN, LH601_MAN := STLV59_563.STLV59_A_563_004.LH601_MAN, LC601_SP := STLV59_563.STLV59_A_563_004.LC601_SP, LC601_MAN := STLV59_563.STLV59_A_563_004.LC601_MAN);
STLV59_563.STLV59_A_563_004.OPM_CV := Rom_004.OPM_CV;
STLV59_563.STLV59_A_563_004.RT601_CS := Rom_004.RT601_CS;
STLV59_563.STLV59_A_563_004.RY600_CV := Rom_004.RY600_CV;
STLV59_563.STLV59_A_563_004.RY600_OP := Rom_004.RY600_OP;
STLV59_563.STLV59_A_563_004.LH601_OP := Rom_004.LH601_OP;
STLV59_563.STLV59_A_563_004.LH601_CMD := Rom_004.LH601_CMD;
STLV59_563.STLV59_A_563_004.LC601_OP := Rom_004.LC601_OP;
STLV59_563.STLV59_A_563_004.LC601_CMD := Rom_004.LC601_CMD;
(* Rom 005 *)
Rom_005(RB601_HVAC := STLV59_563.STLV59_A_563_005.RB601_HVAC, RT601_CT := STLV59_563.STLV59_A_563_005.RT601_CT, RT601_SP_D := STLV59_563.STLV59_A_563_005.RT601_SP_D, RT601_SP_S := STLV59_563.STLV59_A_563_005.RT601_SP_S, RT601_SP_N := STLV59_563.STLV59_A_563_005.RT601_SP_N, RT601_SP_F := STLV59_563.STLV59_A_563_005.RT601_SP_F, OPM := STLV59_563.STLV59_A_563_005.OPM, RY601_CV := STLV59_563.STLV59_A_563_005.RY601_CV, RY601_SP := STLV59_563.STLV59_A_563_005.RY601_SP, RY601_MAN := STLV59_563.STLV59_A_563_005.RY601_MAN, LH601_MAN := STLV59_563.STLV59_A_563_005.LH601_MAN, LC601_SP := STLV59_563.STLV59_A_563_005.LC601_SP, LC601_MAN := STLV59_563.STLV59_A_563_005.LC601_MAN);
STLV59_563.STLV59_A_563_005.OPM_CV := Rom_005.OPM_CV;
STLV59_563.STLV59_A_563_005.RT601_CS := Rom_005.RT601_CS;
STLV59_563.STLV59_A_563_005.RY601_OP := Rom_005.RY601_OP;
STLV59_563.STLV59_A_563_005.LH601_OP := Rom_005.LH601_OP;
STLV59_563.STLV59_A_563_005.LH602_OP := Rom_005.LH602_OP;
STLV59_563.STLV59_A_563_005.LH601_CMD := Rom_005.LH601_CMD;
STLV59_563.STLV59_A_563_005.LC601_OP := Rom_005.LC601_OP;
STLV59_563.STLV59_A_563_005.LC601_CMD := Rom_005.LC601_CMD;
(* Rom 006 *)
Rom_006(RB601_HVAC := STLV59_563.STLV59_A_563_006.RB601_HVAC, RT601_CT := STLV59_563.STLV59_A_563_006.RT601_CT, RT601_SP_D := STLV59_563.STLV59_A_563_006.RT601_SP_D, RT601_SP_S := STLV59_563.STLV59_A_563_006.RT601_SP_S, RT601_SP_N := STLV59_563.STLV59_A_563_006.RT601_SP_N, RT601_SP_F := STLV59_563.STLV59_A_563_006.RT601_SP_F, OPM := STLV59_563.STLV59_A_563_006.OPM, RY601_CV := STLV59_563.STLV59_A_563_006.RY601_CV, RY601_SP := STLV59_563.STLV59_A_563_006.RY601_SP, RY601_MAN := STLV59_563.STLV59_A_563_006.RY601_MAN, LH601_MAN := STLV59_563.STLV59_A_563_006.LH601_MAN, LC601_SP := STLV59_563.STLV59_A_563_006.LC601_SP, LC601_MAN := STLV59_563.STLV59_A_563_006.LC601_MAN);
STLV59_563.STLV59_A_563_006.OPM_CV := Rom_006.OPM_CV;
STLV59_563.STLV59_A_563_006.RT601_CS := Rom_006.RT601_CS;
STLV59_563.STLV59_A_563_006.RY601_OP := Rom_006.RY601_OP;
STLV59_563.STLV59_A_563_006.LH601_OP := Rom_006.LH601_OP;
STLV59_563.STLV59_A_563_006.LH601_CMD := Rom_006.LH601_CMD;
STLV59_563.STLV59_A_563_006.LH602_CMD := Rom_006.LH602_CMD;
STLV59_563.STLV59_A_563_006.LC601_OP := Rom_006.LC601_OP;
STLV59_563.STLV59_A_563_006.LC601_CMD := Rom_006.LC601_CMD;
(* Rom 007 *)
Rom_007(RB601_HVAC := STLV59_563.STLV59_A_563_007.RB601_HVAC, RT601_CT := STLV59_563.STLV59_A_563_007.RT601_CT, RT601_SP_D := STLV59_563.STLV59_A_563_007.RT601_SP_D, RT601_SP_S := STLV59_563.STLV59_A_563_007.RT601_SP_S, RT601_SP_N := STLV59_563.STLV59_A_563_007.RT601_SP_N, RT601_SP_F := STLV59_563.STLV59_A_563_007.RT601_SP_F, OPM := STLV59_563.STLV59_A_563_007.OPM, RY601_CV := STLV59_563.STLV59_A_563_007.RY601_CV, RY601_SP := STLV59_563.STLV59_A_563_007.RY601_SP, RY601_MAN := STLV59_563.STLV59_A_563_007.RY601_MAN, LH601_MAN := STLV59_563.STLV59_A_563_007.LH601_MAN, LC601_SP := STLV59_563.STLV59_A_563_007.LC601_SP, LC601_MAN := STLV59_563.STLV59_A_563_007.LC601_MAN);
STLV59_563.STLV59_A_563_007.OPM_CV := Rom_007.OPM_CV;
STLV59_563.STLV59_A_563_007.RT601_CS := Rom_007.RT601_CS;
STLV59_563.STLV59_A_563_007.RY601_OP := Rom_007.RY601_OP;
STLV59_563.STLV59_A_563_007.LH601_OP := Rom_007.LH601_OP;
STLV59_563.STLV59_A_563_007.LH601_CMD := Rom_007.LH601_CMD;
STLV59_563.STLV59_A_563_007.LC601_OP := Rom_007.LC601_OP;
STLV59_563.STLV59_A_563_007.LC602_OP := Rom_007.LC602_OP;
STLV59_563.STLV59_A_563_007.LC601_CMD := Rom_007.LC601_CMD;
(* Rom 008 *)
Rom_008(RB601_HVAC := STLV59_563.STLV59_A_563_008.RB601_HVAC, RT601_CT := STLV59_563.STLV59_A_563_008.RT601_CT, RT601_SP_D := STLV59_563.STLV59_A_563_008.RT601_SP_D, RT601_SP_S := STLV59_563.STLV59_A_563_008.RT601_SP_S, RT601_SP_N := STLV59_563.STLV59_A_563_008.RT601_SP_N, RT601_SP_F := STLV59_563.STLV59_A_563_008.RT601_SP_F, OPM := STLV59_563.STLV59_A_563_008.OPM, RY601_CV := STLV59_563.STLV59_A_563_008.RY601_CV, RY601_SP := STLV59_563.STLV59_A_563_008.RY601_SP, RY601_MAN := STLV59_563.STLV59_A_563_008.RY601_MAN, LH601_MAN := STLV59_563.STLV59_A_563_008.LH601_MAN, LC601_SP := STLV59_563.STLV59_A_563_008.LC601_SP, LC601_MAN := STLV59_563.STLV59_A_563_008.LC601_MAN);
STLV59_563.STLV59_A_563_008.OPM_CV := Rom_008.OPM_CV;
STLV59_563.STLV59_A_563_008.RT601_CS := Rom_008.RT601_CS;
STLV59_563.STLV59_A_563_008.RY601_OP := Rom_008.RY601_OP;
STLV59_563.STLV59_A_563_008.LH601_OP := Rom_008.LH601_OP;
STLV59_563.STLV59_A_563_008.LH601_CMD := Rom_008.LH601_CMD;
STLV59_563.STLV59_A_563_008.LC601_OP := Rom_008.LC601_OP;
STLV59_563.STLV59_A_563_008.LC601_CMD := Rom_008.LC601_CMD;
STLV59_563.STLV59_A_563_008.LC602_CMD := Rom_008.LC602_CMD;
(* Rom 009 *)
Rom_009(RB601_HVAC := STLV59_563.STLV59_A_563_009.RB601_HVAC, RT601_CT := STLV59_563.STLV59_A_563_009.RT601_CT, RT602_CT := STLV59_563.STLV59_A_563_009.RT602_CT, RT600_SP_D := STLV59_563.STLV59_A_563_009.RT600_SP_D, RT600_SP_S := STLV59_563.STLV59_A_563_009.RT600_SP_S, RT600_SP_N := STLV59_563.STLV59_A_563_009.RT600_SP_N, RT600_SP_F := STLV59_563.STLV59_A_563_009.RT600_SP_F, OPM := STLV59_563.STLV59_A_563_009.OPM, RY601_CV := STLV59_563.STLV59_A_563_009.RY601_CV, RY601_SP := STLV59_563.STLV59_A_563_009.RY601_SP, RY601_MAN := STLV59_563.STLV59_A_563_009.RY601_MAN, LH600_MAN := STLV59_563.STLV59_A_563_009.LH601_MAN, LC600_SP := STLV59_563.STLV59_A_563_009.LC601_SP, LC600_MAN := STLV59_563.STLV59_A_563_009.LC601_MAN);
STLV59_563.STLV59_A_563_009.OPM_CV := Rom_009.OPM_CV;
STLV59_563.STLV59_A_563_009.RT600_CT := Rom_009.RT600_CT;
STLV59_563.STLV59_A_563_009.RT600_CS := Rom_009.RT600_CS;
STLV59_563.STLV59_A_563_009.RY601_OP := Rom_009.RY601_OP;
STLV59_563.STLV59_A_563_009.LH601_OP := Rom_009.LH601_OP;
STLV59_563.STLV59_A_563_009.LH602_OP := Rom_009.LH602_OP;
STLV59_563.STLV59_A_563_009.LH601_CMD := Rom_009.LH601_CMD;
STLV59_563.STLV59_A_563_009.LC601_OP := Rom_009.LC601_OP;
STLV59_563.STLV59_A_563_009.LC601_CMD := Rom_009.LC601_CMD;
(* Rom 010 *)
Rom_010(RB601_HVAC := STLV59_563.STLV59_A_563_010.RB601_HVAC, RT601_CT := STLV59_563.STLV59_A_563_010.RT601_CT, RT602_CT := STLV59_563.STLV59_A_563_010.RT602_CT, RT600_SP_D := STLV59_563.STLV59_A_563_010.RT600_SP_D, RT600_SP_S := STLV59_563.STLV59_A_563_010.RT600_SP_S, RT600_SP_N := STLV59_563.STLV59_A_563_010.RT600_SP_N, RT600_SP_F := STLV59_563.STLV59_A_563_010.RT600_SP_F, OPM := STLV59_563.STLV59_A_563_010.OPM, RY601_CV := STLV59_563.STLV59_A_563_010.RY601_CV, RY601_SP := STLV59_563.STLV59_A_563_010.RY601_SP, RY601_MAN := STLV59_563.STLV59_A_563_010.RY601_MAN, LH600_MAN := STLV59_563.STLV59_A_563_010.LH601_MAN, LC600_SP := STLV59_563.STLV59_A_563_010.LC601_SP, LC600_MAN := STLV59_563.STLV59_A_563_010.LC601_MAN);
STLV59_563.STLV59_A_563_010.OPM_CV := Rom_010.OPM_CV;
STLV59_563.STLV59_A_563_010.RT600_CT := Rom_010.RT600_CT;
STLV59_563.STLV59_A_563_010.RT600_CS := Rom_010.RT600_CS;
STLV59_563.STLV59_A_563_010.RY601_OP := Rom_010.RY601_OP;
STLV59_563.STLV59_A_563_010.LH601_OP := Rom_010.LH601_OP;
STLV59_563.STLV59_A_563_010.LH601_CMD := Rom_010.LH601_CMD;
STLV59_563.STLV59_A_563_010.LH602_CMD := Rom_010.LH602_CMD;
STLV59_563.STLV59_A_563_010.LC601_OP := Rom_010.LC601_OP;
STLV59_563.STLV59_A_563_010.LC601_CMD := Rom_010.LC601_CMD;
(* Rom 011 *)
Rom_011(RB601_HVAC := STLV59_563.STLV59_A_563_011.RB601_HVAC, RT601_CT := STLV59_563.STLV59_A_563_011.RT601_CT, RT602_CT := STLV59_563.STLV59_A_563_011.RT602_CT, RT600_SP_D := STLV59_563.STLV59_A_563_011.RT600_SP_D, RT600_SP_S := STLV59_563.STLV59_A_563_011.RT600_SP_S, RT600_SP_N := STLV59_563.STLV59_A_563_011.RT600_SP_N, RT600_SP_F := STLV59_563.STLV59_A_563_011.RT600_SP_F, OPM := STLV59_563.STLV59_A_563_011.OPM, RY601_CV := STLV59_563.STLV59_A_563_011.RY601_CV, RY601_SP := STLV59_563.STLV59_A_563_011.RY601_SP, RY601_MAN := STLV59_563.STLV59_A_563_011.RY601_MAN, LH600_MAN := STLV59_563.STLV59_A_563_011.LH601_MAN, LC600_SP := STLV59_563.STLV59_A_563_011.LC601_SP, LC600_MAN := STLV59_563.STLV59_A_563_011.LC601_MAN);
STLV59_563.STLV59_A_563_011.OPM_CV := Rom_011.OPM_CV;
STLV59_563.STLV59_A_563_011.RT600_CT := Rom_011.RT600_CT;
STLV59_563.STLV59_A_563_011.RT600_CS := Rom_011.RT600_CS;
STLV59_563.STLV59_A_563_011.RY601_OP := Rom_011.RY601_OP;
STLV59_563.STLV59_A_563_011.LH601_OP := Rom_011.LH601_OP;
STLV59_563.STLV59_A_563_011.LH601_CMD := Rom_011.LH601_CMD;
STLV59_563.STLV59_A_563_011.LC601_OP := Rom_011.LC601_OP;
STLV59_563.STLV59_A_563_011.LC602_OP := Rom_011.LC602_OP;
STLV59_563.STLV59_A_563_011.LC601_CMD := Rom_011.LC601_CMD;
(* Rom 012 *)
Rom_012(RB601_HVAC := STLV59_563.STLV59_A_563_012.RB601_HVAC, RT601_CT := STLV59_563.STLV59_A_563_012.RT601_CT, RT602_CT := STLV59_563.STLV59_A_563_012.RT602_CT, RT600_SP_D := STLV59_563.STLV59_A_563_012.RT600_SP_D, RT600_SP_S := STLV59_563.STLV59_A_563_012.RT600_SP_S, RT600_SP_N := STLV59_563.STLV59_A_563_012.RT600_SP_N, RT600_SP_F := STLV59_563.STLV59_A_563_012.RT600_SP_F, OPM := STLV59_563.STLV59_A_563_012.OPM, RY601_CV := STLV59_563.STLV59_A_563_012.RY601_CV, RY601_SP := STLV59_563.STLV59_A_563_012.RY601_SP, RY601_MAN := STLV59_563.STLV59_A_563_012.RY601_MAN, LH600_MAN := STLV59_563.STLV59_A_563_012.LH601_MAN, LC600_SP := STLV59_563.STLV59_A_563_012.LC601_SP, LC600_MAN := STLV59_563.STLV59_A_563_012.LC601_MAN);
STLV59_563.STLV59_A_563_012.OPM_CV := Rom_012.OPM_CV;
STLV59_563.STLV59_A_563_012.RT600_CT := Rom_012.RT600_CT;
STLV59_563.STLV59_A_563_012.RT600_CS := Rom_012.RT600_CS;
STLV59_563.STLV59_A_563_012.RY601_OP := Rom_012.RY601_OP;
STLV59_563.STLV59_A_563_012.LH601_OP := Rom_012.LH601_OP;
STLV59_563.STLV59_A_563_012.LH601_CMD := Rom_012.LH601_CMD;
STLV59_563.STLV59_A_563_012.LC601_OP := Rom_012.LC601_OP;
STLV59_563.STLV59_A_563_012.LC601_CMD := Rom_012.LC601_CMD;
STLV59_563.STLV59_A_563_012.LC602_CMD := Rom_012.LC602_CMD;
(* Rom 013 *)
Rom_013(RB601_HVAC := STLV59_563.STLV59_A_563_013.RB601_HVAC, RT601_CT := STLV59_563.STLV59_A_563_013.RT601_CT, RT602_CT := STLV59_563.STLV59_A_563_013.RT602_CT, RT600_SP_D := STLV59_563.STLV59_A_563_013.RT600_SP_D, RT600_SP_S := STLV59_563.STLV59_A_563_013.RT600_SP_S, RT600_SP_N := STLV59_563.STLV59_A_563_013.RT600_SP_N, RT600_SP_F := STLV59_563.STLV59_A_563_013.RT600_SP_F, OPM := STLV59_563.STLV59_A_563_013.OPM, RY601_CV := STLV59_563.STLV59_A_563_013.RY601_CV, RY602_CV := STLV59_563.STLV59_A_563_013.RY602_CV, RY600_SP := STLV59_563.STLV59_A_563_013.RY600_SP, RY600_MAN := STLV59_563.STLV59_A_563_013.RY600_MAN, LH600_MAN := STLV59_563.STLV59_A_563_013.LH601_MAN, LC600_SP := STLV59_563.STLV59_A_563_013.LC601_SP, LC600_MAN := STLV59_563.STLV59_A_563_013.LC601_MAN);
STLV59_563.STLV59_A_563_013.OPM_CV := Rom_013.OPM_CV;
STLV59_563.STLV59_A_563_013.RT600_CT := Rom_013.RT600_CT;
STLV59_563.STLV59_A_563_013.RT600_CS := Rom_013.RT600_CS;
STLV59_563.STLV59_A_563_013.RY600_CV := Rom_013.RY600_CV;
STLV59_563.STLV59_A_563_013.RY600_OP := Rom_013.RY600_OP;
STLV59_563.STLV59_A_563_013.LH601_OP := Rom_013.LH601_OP;
STLV59_563.STLV59_A_563_013.LH601_CMD := Rom_013.LH601_CMD;
STLV59_563.STLV59_A_563_013.LC601_OP := Rom_013.LC601_OP;
STLV59_563.STLV59_A_563_013.LC601_CMD := Rom_013.LC601_CMD;
(* Rom 014 *)
Rom_014(RB601_HVAC := STLV59_563.STLV59_A_563_014.RB601_HVAC, RT601_CT := STLV59_563.STLV59_A_563_014.RT601_CT, RT602_CT := STLV59_563.STLV59_A_563_014.RT602_CT, RT600_SP_D := STLV59_563.STLV59_A_563_014.RT600_SP_D, RT600_SP_S := STLV59_563.STLV59_A_563_014.RT600_SP_S, RT600_SP_N := STLV59_563.STLV59_A_563_014.RT600_SP_N, RT600_SP_F := STLV59_563.STLV59_A_563_014.RT600_SP_F, OPM := STLV59_563.STLV59_A_563_014.OPM, RY601_CV := STLV59_563.STLV59_A_563_014.RY601_CV, RY602_CV := STLV59_563.STLV59_A_563_014.RY602_CV, RY600_SP := STLV59_563.STLV59_A_563_014.RY600_SP, RY600_MAN := STLV59_563.STLV59_A_563_014.RY600_MAN, LH600_MAN := STLV59_563.STLV59_A_563_014.LH601_MAN, LC600_SP := STLV59_563.STLV59_A_563_014.LC601_SP, LC600_MAN := STLV59_563.STLV59_A_563_014.LC601_MAN);
STLV59_563.STLV59_A_563_014.OPM_CV := Rom_014.OPM_CV;
STLV59_563.STLV59_A_563_014.RT600_CT := Rom_014.RT600_CT;
STLV59_563.STLV59_A_563_014.RT600_CS := Rom_014.RT600_CS;
STLV59_563.STLV59_A_563_014.RY600_CV := Rom_014.RY600_CV;
STLV59_563.STLV59_A_563_014.RY600_OP := Rom_014.RY600_OP;
STLV59_563.STLV59_A_563_014.LH601_OP := Rom_014.LH601_OP;
STLV59_563.STLV59_A_563_014.LH602_OP := Rom_014.LH602_OP;
STLV59_563.STLV59_A_563_014.LH601_CMD := Rom_014.LH601_CMD;
STLV59_563.STLV59_A_563_014.LH602_CMD := Rom_014.LH602_CMD;
STLV59_563.STLV59_A_563_014.LC601_OP := Rom_014.LC601_OP;
STLV59_563.STLV59_A_563_014.LC602_OP := Rom_014.LC602_OP;
STLV59_563.STLV59_A_563_014.LC601_CMD := Rom_014.LC601_CMD;
STLV59_563.STLV59_A_563_014.LC602_CMD := Rom_014.LC602_CMD;
(* Rom 015 *)
Rom_015(RB601_HVAC := STLV59_563.STLV59_A_563_015.RB601_HVAC, RB602_HVAC := STLV59_563.STLV59_A_563_015.RB602_HVAC, RT601_CT := STLV59_563.STLV59_A_563_015.RT601_CT, RT602_CT := STLV59_563.STLV59_A_563_015.RT602_CT, RT600_SP_D := STLV59_563.STLV59_A_563_015.RT600_SP_D, RT600_SP_S := STLV59_563.STLV59_A_563_015.RT600_SP_S, RT600_SP_N := STLV59_563.STLV59_A_563_015.RT600_SP_N, RT600_SP_F := STLV59_563.STLV59_A_563_015.RT600_SP_F, OPM := STLV59_563.STLV59_A_563_015.OPM, RY601_CV := STLV59_563.STLV59_A_563_015.RY601_CV, RY602_CV := STLV59_563.STLV59_A_563_015.RY602_CV, RY600_SP := STLV59_563.STLV59_A_563_015.RY600_SP, RY600_MAN := STLV59_563.STLV59_A_563_015.RY600_MAN, LH600_MAN := STLV59_563.STLV59_A_563_015.LH601_MAN, LC600_SP := STLV59_563.STLV59_A_563_015.LC601_SP, LC600_MAN := STLV59_563.STLV59_A_563_015.LC601_MAN);
STLV59_563.STLV59_A_563_015.RB600_HVAC := Rom_015.RB600_HVAC;
STLV59_563.STLV59_A_563_015.OPM_CV := Rom_015.OPM_CV;
STLV59_563.STLV59_A_563_015.RT600_CT := Rom_015.RT600_CT;
STLV59_563.STLV59_A_563_015.RT600_CS := Rom_015.RT600_CS;
STLV59_563.STLV59_A_563_015.RY600_CV := Rom_015.RY600_CV;
STLV59_563.STLV59_A_563_015.RY600_OP := Rom_015.RY600_OP;
STLV59_563.STLV59_A_563_015.LH601_OP := Rom_015.LH601_OP;
STLV59_563.STLV59_A_563_015.LH602_OP := Rom_015.LH602_OP;
STLV59_563.STLV59_A_563_015.LH601_CMD := Rom_015.LH601_CMD;
STLV59_563.STLV59_A_563_015.LH602_CMD := Rom_015.LH602_CMD;
STLV59_563.STLV59_A_563_015.LC601_OP := Rom_015.LC601_OP;
STLV59_563.STLV59_A_563_015.LC602_OP := Rom_015.LC602_OP;
STLV59_563.STLV59_A_563_015.LC601_CMD := Rom_015.LC601_CMD;
STLV59_563.STLV59_A_563_015.LC602_CMD := Rom_015.LC602_CMD;
(* Rom 016 *)
Rom_016(RB601_HVAC := STLV59_563.STLV59_A_563_016.RB601_HVAC, RB602_HVAC := STLV59_563.STLV59_A_563_016.RB602_HVAC, RY601_CV := STLV59_563.STLV59_A_563_016.RY601_CV, RY602_CV := STLV59_563.STLV59_A_563_016.RY602_CV, RY600_SP := STLV59_563.STLV59_A_563_016.RY600_SP, RY600_MAN := STLV59_563.STLV59_A_563_016.RY600_MAN, LH601_MAN := STLV59_563.STLV59_A_563_016.LH601_MAN, LC601_SP := STLV59_563.STLV59_A_563_016.LC601_SP, LC601_MAN := STLV59_563.STLV59_A_563_016.LC601_MAN);
STLV59_563.STLV59_A_563_016.RB600_HVAC := Rom_016.RB600_HVAC;
STLV59_563.STLV59_A_563_016.RY600_CV := Rom_016.RY600_CV;
STLV59_563.STLV59_A_563_016.RY600_OP := Rom_016.RY600_OP;
STLV59_563.STLV59_A_563_016.LH601_OP := Rom_016.LH601_OP;
STLV59_563.STLV59_A_563_016.LH602_OP := Rom_016.LH602_OP;
STLV59_563.STLV59_A_563_016.LH601_CMD := Rom_016.LH601_CMD;
STLV59_563.STLV59_A_563_016.LH602_CMD := Rom_016.LH602_CMD;
STLV59_563.STLV59_A_563_016.LC601_OP := Rom_016.LC601_OP;
STLV59_563.STLV59_A_563_016.LC602_OP := Rom_016.LC602_OP;
STLV59_563.STLV59_A_563_016.LC601_CMD := Rom_016.LC601_CMD;
STLV59_563.STLV59_A_563_016.LC602_CMD := Rom_016.LC602_CMD;
END_PROGRAM

PROGRAM PRG_360_HVAC

	STLV59_563.STLV59_A_563_RB001_HVAC:=
(
	STLV59_563.STLV59_A_563_001.RB601_HVAC OR
	STLV59_563.STLV59_A_563_002.RB601_HVAC OR
	STLV59_563.STLV59_A_563_002.RB602_HVAC OR
	STLV59_563.STLV59_A_563_003.RB601_HVAC OR
	STLV59_563.STLV59_A_563_004.RB601_HVAC OR
	STLV59_563.STLV59_A_563_005.RB601_HVAC OR
	STLV59_563.STLV59_A_563_006.RB601_HVAC OR
	STLV59_563.STLV59_A_563_007.RB601_HVAC OR
	STLV59_563.STLV59_A_563_008.RB601_HVAC OR
	STLV59_563.STLV59_A_563_009.RB601_HVAC OR
	STLV59_563.STLV59_A_563_010.RB601_HVAC OR
	STLV59_563.STLV59_A_563_011.RB601_HVAC OR
	STLV59_563.STLV59_A_563_012.RB601_HVAC OR
	STLV59_563.STLV59_A_563_013.RB601_HVAC OR
	STLV59_563.STLV59_A_563_014.RB601_HVAC OR
	STLV59_563.STLV59_A_563_015.RB601_HVAC OR
	STLV59_563.STLV59_A_563_015.RB602_HVAC OR
	STLV59_563.STLV59_A_563_016.RB601_HVAC OR
	STLV59_563.STLV59_A_563_016.RB602_HVAC
);
END_PROGRAM
